FUNCTION alg_s_Dinitialized : BOOL
VAR_INPUT
	state: STATE;
END_VAR

alg_s_Dinitialized := (state.dvar_M_HardwareMap) = (elit_initialized);

END_FUNCTION

(* stored: Version 1.1.0.1, ProductVersion 3.1.4022.18
   POU alg_s_Dinitialized: Id {441aa553-80ba-4e6b-b150-6f4a41141b92}, SpecialFunc None *)
